Fanuc KAREL source: FILE_LIST.kl

PROGRAM T
%NOLOCKGROUP
VAR
 v0 : STRING[40]
 v1 : INTEGER
 v2 : INTEGER
 v3 : ARRAY[10] OF STRING[40]
 v4 : INTEGER
 v5 : INTEGER
BEGIN
 FILE_LIST(v0, v1, v2, v3, v4, v5)
END T
